FUNCTION_BLOCK NCI_REF
VAR_INPUT
END_VAR
VAR_OUTPUT
END_VAR
VAR
	PlcToNci AT %Q* : PLCTONC_NCICHANNEL_REF;
	NciToPlc AT %I* : NcToPlc_NciChannel_Ref;
END_VAR

END_FUNCTION_BLOCK

(* stored: Version 1.1.0.1, ProductVersion 3.1.4024.0
   POU NCI_REF: Id {01579470-34d7-42f5-bfd8-dcb7485817e0}, SpecialFunc None *)
